FUNCTION_BLOCK CLS_test
VAR_INPUT
END_VAR
VAR_OUTPUT
END_VAR
VAR
	a : BOOL;
END_VAR

METHOD METH_inference : POINTER TO LREAL
VAR_INPUT
END_VAR
//impl
END_METHOD

END_FUNCTION_BLOCK

(* stored: Version 1.1.0.1, ProductVersion 3.1.4024.12
   POU CLS_test: Id {2c7506b1-78f3-4a12-a532-7be1c8ef9b8e}, SpecialFunc None
   Method METH_inference: Id {95c329df-c5c1-4fd2-bba7-4af5cddc7160} *)
